TYPE T_ProtobufMaxString : STRING(Param.cMaxCharacter + 1); END_TYPE

(* stored: Version 1.1.0.1
   DUT T_ProtobufMaxString: Id {4ace9a96-660f-4e10-8cd0-e7fb19d4fc95} *)
